TEXTLIST TL_TctrlOutSelect
  0 = 'NoSignal'
  1 = 'PWM'
  2 = 'Sign'
  3 = '2step'
   = ''
END_TEXTLIST

(* stored: Version 1.1.0.1, ProductVersion 3.1.4020.12
   TextList TL_TctrlOutSelect: Id {56d54422-4559-40ed-a10b-949d3a04d31e} *)
